PROGRAM Main3
VAR
	Sequence:Sequence3;
	Forces:Forces3;
	Reset:Reset3;
	Faults:Faults3;
	
	nState 			: INT := 0;
	fbPower			: MC_Power;
	powerOutputs 	: ST_McOutputs;
	reset3Done		: BOOL;
	
	fbMoveRelative: MC_MoveRelative;
	bMoveError: BOOL;
	
END_VAR

CASE nState OF
	0:
		fbPower(
			Axis:= GVL_Conveyer.ConveyerAxis, 
			Enable:= TRUE, 
			Enable_Positive:= TRUE, 
			Enable_Negative:= TRUE,  
			Status=> , 
			Busy=> powerOutputs.Busy, 
			Active=> powerOutputs.Active, 
			Error=> powerOutputs.Error, 
			ErrorID=> powerOutputs.ErrorID);
		IF NOT fbPower.Error THEN
			IF fbPower.Status THEN
				nState := 1;
			END_IF	
		ELSE
			nState := 9999;
		END_IF
	
	1:
		Reset(
			Execute := TRUE,
			bResetDone => reset3Done);
		IF reset3Done THEN
			nState := 2;
		END_IF
		IF Reset.bResetError THEN
			nState := 9999;
		END_IF
		
	2:
	
		Sequence();
		IF Sequence.bSequenceError THEN
			nState := 9999;
		END_IF
	
	9999:
		Faults();
END_CASE

END_PROGRAM

(* stored: Version 1.1.0.1, ProductVersion 3.1.4024.11
   POU Main3: Id {48f3aa79-5c81-4de9-a7df-ef8cb0b063c9}, SpecialFunc None *)
